VAR_GLOBAL
	Axis1	: AXIS_REF;
	Axis2	: AXIS_REF;
	
	stAxis1	: ST_AxisInterface;
	stAxis2	: ST_AxisInterface;
	
	fbMotion1	: FB_Motion;
	fbMotion2	: FB_Motion;
	
END_VAR

(* stored: Version 1.1.0.1, ProductVersion 3.1.4022.12
   GVL GVL_Servo: Id {bc0d18a6-57ae-4db4-bb6b-d64e3bdb82e4} *)
